FUNCTION_BLOCK Axis_stop
VAR_INPUT
	Execute_:BOOL;
END_VAR
VAR_OUTPUT
END_VAR
VAR
	AxisStop:MC_Stop;
	trig1: F_TRIG;
END_VAR

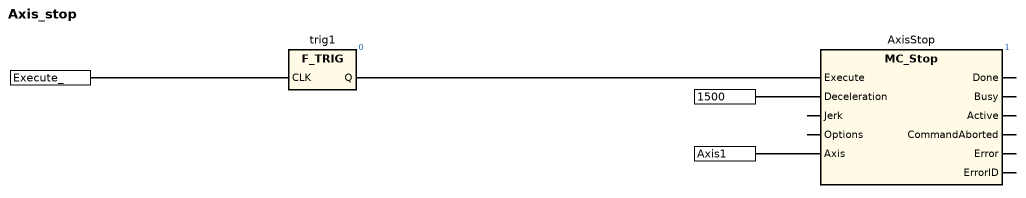
trig1(CLK := Execute_); // F_TRIG
AxisStop(Execute := trig1.Q, Deceleration := 1500, Axis := Axis1); // MC_Stop

END_FUNCTION_BLOCK

(* stored: Version 1.1.0.1, ProductVersion 3.1.4024.12
   POU Axis_stop: Id {c1c1e505-210a-44de-887c-6563451bc73a}, SpecialFunc None *)
